ORGANIZATION_BLOCK OB 100
BEGIN
	L		0
	T		MW 0
	T		AB 8
END_ORGANIZATION_BLOCK


ORGANIZATION_BLOCK OB 1
BEGIN
	L		MW 0
	L		W#16#1000
	==I
	SPB		STOP

	L		MB 1
	L		W#16#FF
	<>I
	SPB		END


	L		EB 8
	L		AB 8
	XOW		W#16#FF
	__ASSERT==	__ACCU 1,	__ACCU 2


END:	L		MW 0
	+		1
	T		MW 0

	L		MB 0
	T		AB 8
	BEA

STOP:	CALL SFC 46 // STOP CPU

END_ORGANIZATION_BLOCK
